// TIA Portal V18 export
FUNCTION "tod_add" : Void   // FC1, FBD
{ S7_Optimized_Access := 'TRUE' }
VERSION : 0.1
// stored: AutoNumber true, IsIECCheckEnabled false, SetENOAutomatically false, UDAEnableTagReadback false
   VAR_INPUT
      i_actualDTL : DTL;
      i_TOD : Time_Of_Day;
      i_TIME : Time;
   END_VAR
   VAR_OUTPUT
      o_TOD : Time_Of_Day;
   END_VAR
   VAR_TEMP
      tempDate : Date;
      tempDTL : DTL;
      tempDTL_1 : DTL;
   END_VAR
   VAR_TEMP   // added for the SCL form of the ladder/FBD networks
      _w1 : Bool;
      _w2 : Bool;
      _w3 : Bool;
   END_VAR
BEGIN

REGION Network 1: TOD add time(over midnight possible)
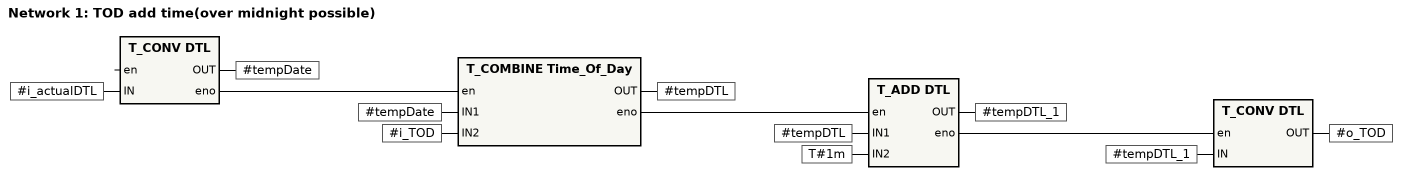
   T_CONV(IN := #i_actualDTL, OUT => #tempDate, ENO => #_w1);
   T_COMBINE(EN := #_w1, IN1 := #tempDate, IN2 := #i_TOD, OUT => #tempDTL, ENO => #_w2);
   T_ADD(EN := #_w2, IN1 := #tempDTL, IN2 := T#1m, OUT => #tempDTL_1, ENO => #_w3);
   IF #_w3 THEN T_CONV(IN := #tempDTL_1, OUT => #o_TOD); END_IF;
END_REGION
END_FUNCTION
